// TIA Portal V20 export
DATA_BLOCK "Data_From_Safety"   // DB4
{ S7_Optimized_Access := 'TRUE' }
// stored: MemoryReserve 100
   VAR
      Safety_Active : Bool;
      Safety_SSP : Bool;
      SSP_R1_1 : Bool;
      SSP_R1_2 : Bool;
      SSP_R2_1 : Bool;
      SSP_R2_2 : Bool;
      PLC_Curing_Safety : Bool;
   END_VAR
BEGIN
END_DATA_BLOCK
